{attribute 'GeneratedUsingTerminal: BK1120-0000-0017'}
{attribute addProperty BoxType "BK1120-0000-0017"}
{attribute addProperty Id "Term_377_KL1002KL1002_BB38DA8F0"}
{attribute addProperty CRC "3685663631"}
{attribute addProperty Size "0"}
TYPE A_0004_BK1120_0000_0017_DBAEC38F EXTENDS BK1120_AEEC0900 :
STRUCT
	{attribute addProperty Name "Term_377_KL1002"}
	Term_377_KL1002 : KL1002_BB38DA8F;
END_STRUCT
END_TYPE

(* stored: Version 1.2.0.0, ProductVersion 3.1.4024.9
   DUT A_0004_BK1120_0000_0017_DBAEC38F: Id {d9037173-d737-44d0-8c08-e42ad4c91db5} *)
